// TIA Portal V17 export
// export: Created 2022-05-25T12:34:01.5515403Z, ExportSetting WithDefaults, DisplayName Totally Integrated Automation Portal, DisplayVersion V17, DisplayName TIA Portal Openness, DisplayVersion V17, DisplayName TIA Portal Version Control Interface, DisplayVersion V17, DisplayName STEP 7 Professional, DisplayVersion V17, DisplayName STEP 7 Safety, DisplayVersion V17, DisplayName WinCC Professional, DisplayVersion V17
VAR_GLOBAL   // PLC tag table "GP25_Yaskawa_Input_Mapping"
   External_Start AT %Q3192.0 : Bool;
   External_Servo_On AT %Q3192.1 : Bool;
   Call_Master_Job AT %Q3192.2 : Bool;
   Alarm_Reset AT %Q3192.3 : Bool;
   Reduced_Speed AT %Q3192.4 : Bool;
   Buzzer AT %Q3192.5 : Bool;
   Watchdog AT %Q3192.6 : Bool;
   Lowe_Air_Pressure AT %Q3192.7 : Bool;
   Machine_Lock AT %Q3193.0 : Bool;
   Reserve_System_Area AT %Q3193.1 : Bool;
   External_Hold AT %Q3193.2 : Bool;
   Invalid_Collision_Detect AT %Q3193.3 : Bool;
   Continues_Cycle_Select AT %Q3193.4 : Bool;
   "1_Cycle_Select" AT %Q3193.5 : Bool;
   Edit_Lock AT %Q3193.6 : Bool;
   Auto_Backup AT %Q3193.7 : Bool;
   Work_Prohibite_R1 AT %Q3194.0 : Bool;
   Work_Prohibite_R2 AT %Q3194.1 : Bool;
   Work_Prohibite_R3 AT %Q3194.2 : Bool;
   Work_Prohibite_R4 AT %Q3194.3 : Bool;
   Work_Prohibite_R5 AT %Q3194.4 : Bool;
   Work_Prohibite_R6 AT %Q3194.5 : Bool;
   Work_Prohibite_R7 AT %Q3194.6 : Bool;
   Work_Prohibite_R8 AT %Q3194.7 : Bool;
   Secuence_Wait_R1 AT %Q3195.0 : Bool;
   Secuence_Wait_R2 AT %Q3195.1 : Bool;
   Secuence_Wait_R3 AT %Q3195.2 : Bool;
   Secuence_Wait_R4 AT %Q3195.3 : Bool;
   Secuence_Wait_R5 AT %Q3195.4 : Bool;
   Secuence_Wait_R6 AT %Q3195.5 : Bool;
   Secuence_Wait_R7 AT %Q3195.6 : Bool;
   Secuence_Wait_R8 AT %Q3195.7 : Bool;
   Secuence_Wait_S1 AT %Q3196.0 : Bool;
   Secuence_Wait_S2 AT %Q3196.1 : Bool;
   Secuence_Wait_S3 AT %Q3196.2 : Bool;
   Secuence_Wait_S4 AT %Q3196.3 : Bool;
   Secuence_Wait_S5 AT %Q3196.4 : Bool;
   Secuence_Wait_S6 AT %Q3196.5 : Bool;
   Secuence_Wait_S7 AT %Q3196.6 : Bool;
   Secuence_Wait_S8 AT %Q3196.7 : Bool;
   STATUS_BIT_0 AT %Q3191.0 : Bool;
   STATUS_BIT_1 AT %Q3191.1 : Bool;
   STATUS_BIT_2 AT %Q3191.2 : Bool;
   STATUS_BIT_3 AT %Q3191.3 : Bool;
   STATUS_BIT_4 AT %Q3191.4 : Bool;
   STATUS_BIT_5 AT %Q3191.5 : Bool;   // IF = 1 Some Slaves are unreachable
   STATUS_BIT_6 AT %Q3191.6 : Bool;   // IF = 1 All Slaves are unreachable
   STATUS_BIT_7 AT %Q3191.7 : Bool;   // IF = 1 Master is unreachable
   Step_Back_R1 AT %Q3197.0 : Bool;
   Step_Back_R2 AT %Q3197.1 : Bool;
   Step_Back_R3 AT %Q3197.2 : Bool;
   Step_Back_R4 AT %Q3197.3 : Bool;
   Step_Back_R5 AT %Q3197.4 : Bool;
   Step_Back_R6 AT %Q3197.5 : Bool;
   Step_Back_R7 AT %Q3197.6 : Bool;
   Step_Back_R8 AT %Q3197.7 : Bool;
   Extern_Servo_Off_Hold_Stop AT %Q3198.0 : Bool;
   Extern_Servo_OFF_2 AT %Q3198.1 : Bool;   // E_STOP CATEGORY 0
   Extern_Servo_OFF_3 AT %Q3198.2 : Bool;   // E_STOP CATEGORY 1
END_VAR
